% RSLogix 500 project I2P Job 07 - Andrew_Hoemmen.RSS, saved by version 10.00.00.00 %
PROJECT "ML03A"    % processor: Bul.1763 MicroLogix 1100 Series B %

PROGRAM FILES
  LAD 2   3 rungs

DATA FILES
  O0 OUTPUT  4 elements
  I1 INPUT  6 elements
  S2 STATUS  66 elements
  B3 BINARY  1 elements
  T4 TIMER  1 elements
  C5 COUNTER  1 elements
  R6 CONTROL  1 elements
  N7 INTEGER  1 elements
  F8 FLOAT  1 elements

LADDER 2
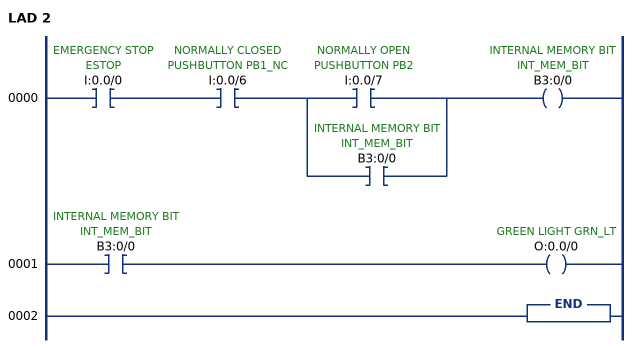
% Rung: 0 %
SOR XIC I:0.0/0 XIC I:0.0/6 BST XIC I:0.0/7 NXB XIC B3:0/0 BND OTE B3:0/0 EOR
%   I:0.0/0  ESTOP  "EMERGENCY STOP" %
%   I:0.0/6  PB1_NC  "NORMALLY CLOSED PUSHBUTTON" %
%   I:0.0/7  PB2  "NORMALLY OPEN PUSHBUTTON" %
%   B3:0/0  INT_MEM_BIT  "INTERNAL MEMORY BIT" %
% Rung: 1 %
SOR XIC B3:0/0 OTE O:0.0/0 EOR
%   B3:0/0  INT_MEM_BIT  "INTERNAL MEMORY BIT" %
%   O:0.0/0  GRN_LT  "GREEN LIGHT" %
% Rung: 2 %
SOR END EOR

OTHER DOCUMENTED ADDRESSES
  I:0.0/1  CR1_STAT  "CONTROL RELAY 1 CONTACTS"
  I:0.0/2  CR2_STATS  "CONTROL RELAY 2 CONTACTS"
  I:0.0/3  3PSS_A  "THREE POSITION SELECTOR SWITCH A POSITION"
  I:0.0/4  3PSS_B  "THREE POSITION SELECTOR SWITCH B POSITION"
  I:0.0/5  2PSS  "TWO POSITION SELECTOR SWITCH"
  I:0.0/8  PB3  "NORMALLY OPEN PUSHBUTTON"
  O:0.0/1  YEL_LT  "YELLOW LIGHT"
  O:0.0/2  RED_LT  "RED LIGHT"
  O:0.0/3  BLUE_LT  "BLUE LIGHT"
  O:0.0/4  CR1  "CONTROL RELAY 1"
  O:0.0/5  CR2  "CONTROL RELAY 2"
